PROGRAM MAIN
VAR
	vector_2 : ARRAY[0..2] OF LREAL := [1,1,1];	
	out : ARRAY[0..0] OF LREAL;
	FB_NN : FB_Dense_v1;

END_VAR

FB_NN(pointer_input := ADR(vector_2),pointer_output:= ADR(out));
//sum := F_DATA_TO_CRC16_CCITT(pData := ADR(FB_NN.nn.weights),cbData := SIZEOF(FB_NN.nn.weights),crc:=crc);
//sum2 := F_CheckSum16(dwSrcAddr := ADR(FB_NN.nn.weights),cbLen := SIZEOF(FB_NN.nn.weights),wChkSum:=crc);

END_PROGRAM

(* stored: Version 1.1.0.1, ProductVersion 3.1.4024.12
   POU MAIN: Id {5aa131dd-eb33-4156-8cfc-71109cf3c4fe}, SpecialFunc None *)
